(* Gets the lower bound index of :itf:`I_Runnable` array.*)
FUNCTION F_GetRunnableArrayLowerBound : T_Position
VAR_IN_OUT
	arRunnables : ARRAY[*] OF REAL; // The array to query.
END_VAR

F_GetRunnableArrayLowerBound := LOWER_BOUND(arRunnables, 1);

END_FUNCTION

(* stored: Version 1.1.0.1
   POU F_GetRunnableArrayLowerBound: Id {c0a2bbfd-fa17-098b-1d31-6f1edd9b3c20}, SpecialFunc None *)
